PROGRAM NIET_GOED_LEZEN
VAR
END_VAR

END_PROGRAM

(* stored: Version 1.1.0.1, ProductVersion 3.1.4024.15
   POU NIET_GOED_LEZEN: Id {ef78d04c-f904-48ac-b28f-3fe7a5e193ec}, SpecialFunc None *)
